FUNCTION_BLOCK ThreeConCtl (* Composite Function Block Type *)
  (* Standard: 61499-2 *)
  (* Version 0.2, 2003-12-05, JHC, Rockwell Automation, Renamed from NEWCOMPFB. *)
  (* Version 0.1, 2002-01-08, JHC, Rockwell Automation, Added DLY FB as example. *)
  (* Version 0.0, 2000-05-27, JHC, Rockwell Automation *)
  (* Compiler header: package fb.rt.cs725; *)
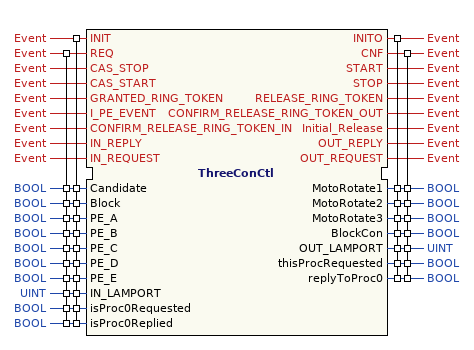
  EVENT_INPUT
    INIT WITH Candidate, Block, PE_A, PE_B, PE_C, PE_D, PE_E, isProc0Requested, IN_LAMPORT, isProc0Replied; (* Initialization Request *)
    REQ WITH Block, Candidate, PE_A, PE_B, PE_C, PE_D, PE_E, IN_LAMPORT, isProc0Requested, isProc0Replied; (* Normal Execution Request *)
    CAS_STOP;
    CAS_START;
    GRANTED_RING_TOKEN;
    I_PE_EVENT;
    CONFIRM_RELEASE_RING_TOKEN_IN;
    IN_REPLY;
    IN_REQUEST;
  END_EVENT
  EVENT_OUTPUT
    INITO WITH MotoRotate1, MotoRotate2, MotoRotate3, BlockCon, thisProcRequested, replyToProc0, OUT_LAMPORT; (* Initialization Confirm *)
    CNF WITH MotoRotate1, MotoRotate2, MotoRotate3, BlockCon, OUT_LAMPORT, thisProcRequested, replyToProc0; (* Execution Confirmation *)
    START;
    STOP;
    RELEASE_RING_TOKEN;
    CONFIRM_RELEASE_RING_TOKEN_OUT;
    Initial_Release;
    OUT_REPLY;
    OUT_REQUEST;
  END_EVENT
  VAR_INPUT
    Candidate : BOOL;
    Block : BOOL;
    PE_A : BOOL;
    PE_B : BOOL;
    PE_C : BOOL;
    PE_D : BOOL;
    PE_E : BOOL;
    IN_LAMPORT : UINT;
    isProc0Requested : BOOL;
    isProc0Replied : BOOL;
  END_VAR
  VAR_OUTPUT
    MotoRotate1 : BOOL;
    MotoRotate2 : BOOL;
    MotoRotate3 : BOOL;
    BlockCon : BOOL;
    OUT_LAMPORT : UINT;
    thisProcRequested : BOOL;
    replyToProc0 : BOOL;
  END_VAR
  FBS
    FC11 : ConveyorRingTokenCTL(HAS_INITIAL_TOKEN := 0);
    FC12 : ConveyorCTLMulticast(Block := 0, Candidate := 0);
    FC13 : ConveyorCTL(Block := 0, Candidate := 0);
  END_FBS
  EVENT_CONNECTIONS
    INIT TO FC11.INIT;
    REQ TO FC11.REQ;
    FC11.INITO TO FC12.INIT;
    FC12.INITO TO FC13.INIT;
    FC13.INITO TO INITO;
    FC13.CNF TO CNF;
    REQ TO FC12.REQ;
    REQ TO FC13.REQ;
    FC11.CNF TO CNF;
    FC12.CNF TO CNF;
    CAS_STOP TO FC11.CAS_STOP;
    CAS_START TO FC11.CAS_START;
    FC13.STOP TO STOP;
    FC13.START TO START;
    I_PE_EVENT TO FC11.I_PE_EVENT;
    CONFIRM_RELEASE_RING_TOKEN_IN TO FC11.CONFIRM_TOKEN_RECEIVED_IN;
    GRANTED_RING_TOKEN TO FC11.GRANTED_RING_TOKEN;
    FC11.RELEASE_RING_TOKEN TO RELEASE_RING_TOKEN;
    FC11.CONFIRM_TOKEN_RECEIVED_OUT TO CONFIRM_RELEASE_RING_TOKEN_OUT;
    CAS_STOP TO FC12.CAS_STOP;
    CAS_START TO FC12.CAS_START;
    I_PE_EVENT TO FC12.PE_EVENT;
    IN_REPLY TO FC12.IN_REPLY;
    IN_REQUEST TO FC12.IN_REQUEST;
    FC12.OUT_REPLY TO OUT_REPLY;
    FC12.OUT_REQUEST TO OUT_REQUEST;
  END_CONNECTIONS
  DATA_CONNECTIONS
    FC13.MotoRotate TO MotoRotate3;
    FC12.MotoRotate TO MotoRotate2;
    FC11.MotoRotate TO MotoRotate1;
    Block TO FC11.Block;
    FC11.BlockCon TO BlockCon;
    Candidate TO FC11.Candidate;
    PE_C TO FC13.PE;
    PE_A TO FC11.PE_IN;
    PE_B TO FC11.PE_OUT;
    PE_D TO FC12.PE_OUT;
    PE_C TO FC12.PE_IN;
    thisProcRequested TO FC12.isProc0Requested;
    isProc0Replied TO FC12.isProc0Replied;
    FC12.thisProcRequested TO thisProcRequested;
    FC12.replyToProc0 TO replyToProc0;
    IN_LAMPORT TO FC12.IN_LAMPORT;
    FC12.OUT_LAMPORT TO OUT_LAMPORT;
  END_CONNECTIONS
END_FUNCTION_BLOCK
